PROGRAM AP_1_1
VAR
	GetPlate			:Seq_Get_Part;
	SetPlate1			:Seq_Set_Plate_1;
	SetPlate2			:Seq_Set_Plate_2;
	AusrichtenPlates 	:Seq_Ausrichten_Plates;
	SetMountingPlate	:Seq_Set_MPlate;
	AusrichtenMP		:Seq_Ausrichten_MPlate;
END_VAR

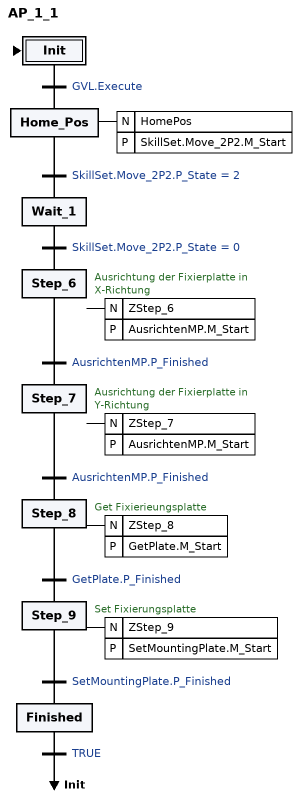
INITIAL_STEP Init:
END_STEP
TRANSITION FROM Init TO Home_Pos
    := GVL.Execute;
END_TRANSITION
STEP Home_Pos:
    HomePos(N);
    SkillSet.Move_2P2.M_Start(P);
END_STEP
TRANSITION FROM Home_Pos TO Wait_1
    := SkillSet.Move_2P2.P_State = 2;
END_TRANSITION
STEP Wait_1:
END_STEP
TRANSITION FROM Wait_1 TO Step_6
    := SkillSet.Move_2P2.P_State = 0;
END_TRANSITION
// Ausrichtung der Fixierplatte in X-Richtung
STEP Step_6:
    ZStep_6(N);
    AusrichtenMP.M_Start(P);
END_STEP
TRANSITION FROM Step_6 TO Step_7
    := AusrichtenMP.P_Finished;
END_TRANSITION
// Ausrichtung der Fixierplatte in Y-Richtung
STEP Step_7:
    ZStep_7(N);
    AusrichtenMP.M_Start(P);
END_STEP
TRANSITION FROM Step_7 TO Step_8
    := AusrichtenMP.P_Finished;
END_TRANSITION
// Get Fixierieungsplatte
STEP Step_8:
    ZStep_8(N);
    GetPlate.M_Start(P);
END_STEP
TRANSITION FROM Step_8 TO Step_9
    := GetPlate.P_Finished;
END_TRANSITION
// Set Fixierungsplatte
STEP Step_9:
    ZStep_9(N);
    SetMountingPlate.M_Start(P);
END_STEP
TRANSITION FROM Step_9 TO Finished
    := SetMountingPlate.P_Finished;
END_TRANSITION
STEP Finished:
END_STEP
TRANSITION FROM Finished TO Init
    := TRUE;
END_TRANSITION

ACTION HomePos:
SkillSet.Move_2P2.P_RobotParam := PunkteZuweisung_Temp.PHome;
END_ACTION

ACTION ZStep_1:
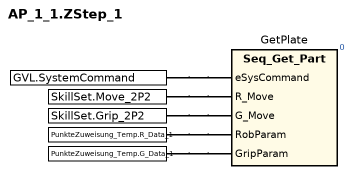
GetPlate(
    eSysCommand := GVL.SystemCommand,
    R_Move := SkillSet.Move_2P2,
    G_Move := SkillSet.Grip_2P2,
    RobParam := PunkteZuweisung_Temp.R_Data_1,
    GripParam := PunkteZuweisung_Temp.G_Data_1); // Seq_Get_Part
END_ACTION

ACTION ZStep_2:
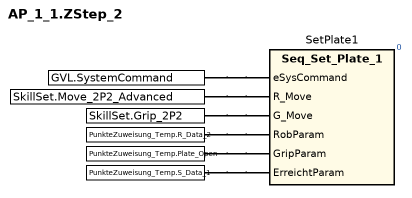
SetPlate1(
    eSysCommand := GVL.SystemCommand,
    R_Move := SkillSet.Move_2P2_Advanced,
    G_Move := SkillSet.Grip_2P2,
    RobParam := PunkteZuweisung_Temp.R_Data_2,
    GripParam := PunkteZuweisung_Temp.Plate_Open,
    ErreichtParam := PunkteZuweisung_Temp.S_Data_1); // Seq_Set_Plate_1
END_ACTION

ACTION ZStep_3:
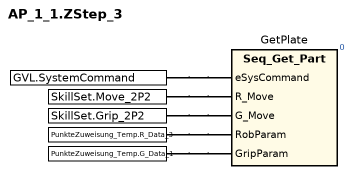
GetPlate(
    eSysCommand := GVL.SystemCommand,
    R_Move := SkillSet.Move_2P2,
    G_Move := SkillSet.Grip_2P2,
    RobParam := PunkteZuweisung_Temp.R_Data_3,
    GripParam := PunkteZuweisung_Temp.G_Data_1); // Seq_Get_Part
END_ACTION

ACTION ZStep_4:
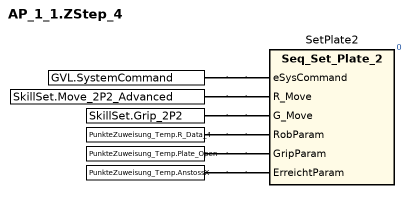
SetPlate2(
    eSysCommand := GVL.SystemCommand,
    R_Move := SkillSet.Move_2P2_Advanced,
    G_Move := SkillSet.Grip_2P2,
    RobParam := PunkteZuweisung_Temp.R_Data_4,
    GripParam := PunkteZuweisung_Temp.Plate_Open,
    ErreichtParam := PunkteZuweisung_Temp.AnstossX); // Seq_Set_Plate_2
END_ACTION

ACTION ZStep_5:
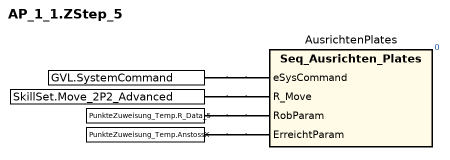
AusrichtenPlates(
    eSysCommand := GVL.SystemCommand,
    R_Move := SkillSet.Move_2P2_Advanced,
    RobParam := PunkteZuweisung_Temp.R_Data_5,
    ErreichtParam := PunkteZuweisung_Temp.AnstossX); // Seq_Ausrichten_Plates
END_ACTION

ACTION ZStep_6:
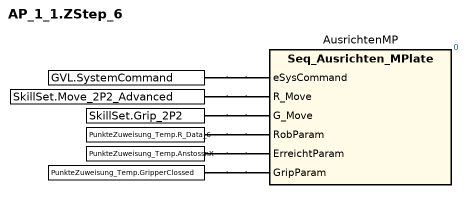
AusrichtenMP(
    eSysCommand := GVL.SystemCommand,
    R_Move := SkillSet.Move_2P2_Advanced,
    G_Move := SkillSet.Grip_2P2,
    RobParam := PunkteZuweisung_Temp.R_Data_6,
    ErreichtParam := PunkteZuweisung_Temp.AnstossnX,
    GripParam := PunkteZuweisung_Temp.GripperClossed); // Seq_Ausrichten_MPlate
END_ACTION

ACTION ZStep_7:
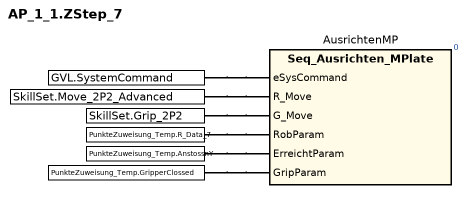
AusrichtenMP(
    eSysCommand := GVL.SystemCommand,
    R_Move := SkillSet.Move_2P2_Advanced,
    G_Move := SkillSet.Grip_2P2,
    RobParam := PunkteZuweisung_Temp.R_Data_7,
    ErreichtParam := PunkteZuweisung_Temp.AnstossnY,
    GripParam := PunkteZuweisung_Temp.GripperClossed); // Seq_Ausrichten_MPlate
END_ACTION

ACTION ZStep_8:
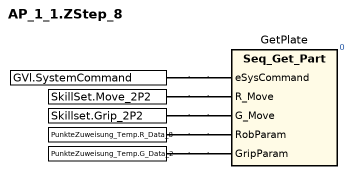
GetPlate(
    eSysCommand := GVl.SystemCommand,
    R_Move := SkillSet.Move_2P2,
    G_Move := Skillset.Grip_2P2,
    RobParam := PunkteZuweisung_Temp.R_Data_8,
    GripParam := PunkteZuweisung_Temp.G_Data_2); // Seq_Get_Part
END_ACTION

ACTION ZStep_9:
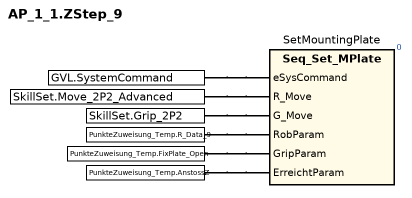
SetMountingPlate(
    eSysCommand := GVL.SystemCommand,
    R_Move := SkillSet.Move_2P2_Advanced,
    G_Move := SkillSet.Grip_2P2,
    RobParam := PunkteZuweisung_Temp.R_Data_9,
    GripParam := PunkteZuweisung_Temp.FixPlate_Open,
    ErreichtParam := PunkteZuweisung_Temp.AnstossZ); // Seq_Set_MPlate
END_ACTION

END_PROGRAM

(* stored: Version 1.1.0.1
   POU AP_1_1: Id {86bb28e9-198f-4bc2-9a63-e1da0719bf32}, SpecialFunc None
   Folder 01_Zuweisung: Id {55f52a54-160d-4fa0-a1ef-bf9cf362354a}
   Action HomePos: Id {3d56fe5e-6953-4e6d-bd63-5e07e2d1f37d}
   Action ZStep_1: Id {23ad8667-829f-4223-9e40-401fbe5b067a}
   Action ZStep_2: Id {27d62ca3-4395-43a7-9080-4cfc3c148be5}
   Action ZStep_3: Id {22dd5a07-d51a-423f-bab9-344fa441fb0e}
   Action ZStep_4: Id {9eae2ba8-5b5d-489e-97cb-773b32c9c977}
   Action ZStep_5: Id {e27c2448-066e-4373-b128-d3a8c834dce2}
   Action ZStep_6: Id {0a07fd20-457f-4cb4-8c99-ea0d2ec44b6b}
   Action ZStep_7: Id {fa6bd752-0bd7-4557-a9ec-84cd3f6f19d3}
   Action ZStep_8: Id {35cd52a2-30bb-49af-aafa-27ef35c05b05}
   Action ZStep_9: Id {9ea02f05-a35c-4ed4-8140-571583e14358} *)
